// TwinCAT 3 PLC project Modbus_RTU
// ProgramVersion: 3.1.4024.12
// libraries:
//   Tc2_ModbusRTU, * (Beckhoff Automation GmbH)
//   Tc2_Standard, * (Beckhoff Automation GmbH)
//   Tc2_System, * (Beckhoff Automation GmbH)
//   Tc3_Module, * (Beckhoff Automation GmbH)
// project tree:
//   / PlcTask.TcTTO
//   POUs/ MAIN.TcPOU, P_ModbusRTU_Master.TcPOU, P_ModbusRTU_Slave.TcPOU

CONFIGURATION Modbus_RTU
    RESOURCE PLC ON TwinCAT3
        TASK PlcTask(INTERVAL := T#10ms, PRIORITY := 28);
        PROGRAM MAIN WITH PlcTask : MAIN;
    END_RESOURCE
END_CONFIGURATION

// ---- POUs/MAIN.TcPOU
PROGRAM MAIN
VAR
END_VAR

P_ModbusRTU_Master();
P_ModbusRTU_Slave();

END_PROGRAM

// ---- POUs/P_ModbusRTU_Master.TcPOU
PROGRAM P_ModbusRTU_Master
VAR
// Communication block
// ===================
	// make sure to choose the correct block depending on the type of serial port
	fbModbus		: ModbusRtuMasterV2_PcCOM;	
	//	fbModbus		: ModbusRtuMasterV2_KL6x5B;	
	//	fbModbus		: ModbusRtuMasterV2_KL6x22B;	
	
// Send and Receive data 
// =====================
	Send			: ARRAY [0..100] OF WORD;
	Rcv				: ARRAY [0..100] OF WORD;

	
// Sequence 
// ========
	bStart			: BOOL;
	Step			: INT;
END_VAR

{region "Hardware set up"}
// Linking to serial port
// ======================

// The IO's to link to the serial port are declared inside of the FB ModbusRtuMasterV2_XXXXX.
// By building/compiling the program, these IO will be generate in the PLC instance, ready to link
// This is also the reason why there are FB's for every type of serial port.

// Communication parameters serial port
// ====================================
	 
// Make sure to set up the correct communication parameters for the serial port, like:
//		* Baudrate
//		* Data bits
//		* Stop bits
//		* Xon/Xoff

// In case you are using an EL terminal, please set these CoE Online parameters:
//		* 	8000:05		"Enable transfer rate opmitization"		--> FALSE
//		*	8000:06		"Enable half duplex"					--> FALSE		(if 4 wires are used for RS485)
//																--> TRUE		(if 2 wires are used for RS485)	 

{endregion}

// Communication block
// ===================

// The communication block itself does not need to be called.
// Depending on the wanted action (read registers, read input registers, write registeres, ...), the corresponding action will be called.
// But since all these actions use the inputs/outputs from the FB itself, it is recommended to use a sequence for calling the actions


// Sequence
// ========

CASE Step OF
	0:		// Wait for start
		IF bStart THEN
			Step := 100;
		END_IF
	100:	// Read input registers 4 - 9 (so 6 modbus registers), from device address 10
		fbModbus.ReadInputRegs(Execute		:= FALSE);		// call actions with "Execute := FALSE", to be sure to have a positive edge to trigger the reading	
		fbModbus.ReadInputRegs(
			UnitID		:= 10, 
			Quantity	:= 6, 
			MBAddr		:= 4,		// Keep in mind that for some devices you have to substract 1 from the register.
			cbLength	:= SIZEOF(Rcv), 
			pMemoryAddr	:= ADR(Rcv), 
			Execute		:= TRUE, 
			Timeout		:= T#100MS,	// Always insert a time out, otherwise a time of 0ms will be used, resulting in a time out  
			BUSY		=> , 
			Error		=> , 
			ErrorId		=> , 
			cbRead		=> );
		
		IF fbModbus.BUSY THEN
			Step := 110;
		END_IF

	110:
		IF NOT fbModbus.BUSY THEN
			IF fbModbus.Error THEN
				// Code to be done in case of an error reading data, f.e.:
				Step := 100;	// if you want to try again
				Step := 0;		// if you want to retry the complete cycle
			ELSE
				// Code to be done in case of no error reading data, f.e.:
				
				// Decode received data
				// Since modbus as a standard only has words, data can be converted to store them in words.
				// for esample, reals are sometimes stored in the words by multiplying them by 10 or by 100, depeding on the wanted resolution
				
				// Reg4Value := Rcv[0] * 0.1;
				// Reg5Value := Rcv[0] * 0.01;
				// Reg6Value := Rcv[0] * 2;
				// Reg7Value := Rcv[0] * 0.1;
				// Reg8Value := Rcv[0] * 0.1;
				// Reg9Value := Rcv[0] * 0.1;
				
				Step := 200;
			END_IF
		END_IF

	200:	// Read registers 12 - 15 (so 4 modbus registers), from device address 15
		fbModbus.ReadRegs(Execute		:= FALSE);		// call actions with "Execute := FALSE", to be sure to have a positive edge to trigger the reading	
		fbModbus.ReadRegs(
			UnitID		:= 15, 
			Quantity	:= 4, 
			MBAddr		:= 12,		// Keep in mind that for some devices you have to substract 1 from the register.
			cbLength	:= SIZEOF(Rcv), 
			pMemoryAddr	:= ADR(Rcv), 
			Execute		:= TRUE, 
			Timeout		:= T#100MS,	// Always insert a time out, otherwise a time of 0ms will be used, resulting in a time out  
			BUSY		=> , 
			Error		=> , 
			ErrorId		=> , 
			cbRead		=> );
		
		IF fbModbus.BUSY THEN
			Step := 210;
		END_IF

	210:
		IF NOT fbModbus.BUSY THEN
			IF fbModbus.Error THEN
				// Code to be done in case of an error reading data, f.e.:
				Step := 200;	// if you want to try again
				Step := 0;		// if you want to retry the complete cycle
			ELSE
				// Code to be done in case of no error reading data, f.e.:
				
				// Decode received data
				// Since modbus as a standard only has words, data can be converted to store them in words.
				// for esample, reals are sometimes stored in the words by multiplying them by 10 or by 100, depeding on the wanted resolution
				
				// Reg12Value := Rcv[0] * 0.1;
				// Reg13Value := Rcv[0] * 0.01;
				// Reg14Value := Rcv[0] * 2;
				// Reg15Value := Rcv[0] * 0.1;
				
				Step := 300;
			END_IF
		END_IF

	300:	// Write registers 25 - 34 (so 10 modbus registers), to device address 27

		// fill data to send:
		Send[0]	:= 1254;		// Data for modbus register 25
		Send[1]	:= 751;			// Data for modbus register 26
		Send[2]	:= 2300;		// Data for modbus register 27
		Send[3]	:= 254;			// Data for modbus register 28
		Send[5]	:= 128;			// Data for modbus register 29
		Send[5]	:= 775;			// Data for modbus register 30
		Send[6]	:= 943;			// Data for modbus register 31
		Send[7]	:= 225;			// Data for modbus register 32
		Send[8].0	:= TRUE;	// Data for modbus register 33
		Send[8].1	:= TRUE;	// Data for modbus register 33
		Send[8].2	:= TRUE;	// Data for modbus register 33
		Send[8].5	:= TRUE;	// Data for modbus register 33
		Send[8].7	:= TRUE;	// Data for modbus register 33
		Send[9]	:= 567;			// Data for modbus register 34
 	
		fbModbus.WriteRegs(Execute		:= FALSE);		// call actions with "Execute := FALSE", to be sure to have a positive edge to trigger the reading	
		fbModbus.WriteRegs(
			UnitID		:= 27, 
			Quantity	:= 10, 
			MBAddr		:= 25,		// Keep in mind that for some devices you have to substract 1 from the register.
			cbLength	:= SIZEOF(Send), 
			pMemoryAddr	:= ADR(Send), 
			Execute		:= TRUE, 
			Timeout		:= T#100MS,	// Always insert a time out, otherwise a time of 0ms will be used, resulting in a time out  
			BUSY		=> , 
			Error		=> , 
			ErrorId		=> , 
			cbRead		=> );
		
		IF fbModbus.BUSY THEN
			Step := 310;
		END_IF

	310:
		IF NOT fbModbus.BUSY THEN
			IF fbModbus.Error THEN
				// Code to be done in case of an error reading data, f.e.:
				Step := 300;	// if you want to try again
				Step := 0;		// if you want to retry the complete cycle
			ELSE
				// Code to be done in case of no error reading data, f.e.:
				
				Step := 0;		// Return to first step
			END_IF
		END_IF
END_CASE

END_PROGRAM

// ---- POUs/P_ModbusRTU_Slave.TcPOU
PROGRAM P_ModbusRTU_Slave
VAR
// Communication block
// ===================
	// make sure to choose the correct block depending on the type of serial port
	fbModbus			: ModbusRtuSlave_PcCOM;	
	//	fbModbus		: ModbusRtuSlave_KL6x5B;	
	//	fbModbus		: ModbusRtuSlave_KL6x22B;	
	
	
// Definition of Modbus data access areas
// ======================================
	// Check the following options *)

	// hardware independent access to the input, output and memory area
	// The ranges are declared with a length of only one word
	// Nevertheless ModbusRTU will access the full length defined above

	(*
	Inputs 	AT %IW0:	WORD;
	Outputs AT %QW0:	WORD;
	Memory 	AT %MW0:	WORD;
	*)

	// The ranges are declared as arrays here (optional)
	Inputs 	AT %IW0:	ARRAY[0..255] OF WORD;
	Outputs AT %QW0:	ARRAY[0..255] OF WORD;
	Memory 	AT %MW0:	ARRAY[0..2047] OF WORD;

	// hardware independent access to normal variables
	// (no input, ouput or memory range)
	
	(*
	Inputs	:	ARRAY[0..255] OF WORD;
	Outputs :	ARRAY[0..255] OF WORD;
	Memory 	:	ARRAY[0..255] OF WORD;
	*)

END_VAR

{region "Hardware set up"}
// Linking to serial port
// ======================

// The IO's to link to the serial port are declared inside of the FB ModbusRtuMasterV2_XXXXX.
// By building/compiling the program, these IO will be generate in the PLC instance, ready to link
// This is also the reason why there are FB's for every type of serial port.

// Communication parameters serial port
// ====================================
	 
// Make sure to set up the correct communication parameters for the serial port, like:
//		* Baudrate
//		* Data bits
//		* Stop bits
//		* Xon/Xoff

// In case you are using an EL terminal, please set these CoE Online parameters:
//		* 	8000:05		"Enable transfer rate opmitization"		--> FALSE
//		*	8000:06		"Enable half duplex"					--> FALSE		(if 4 wires are used for RS485)
//																--> TRUE		(if 2 wires are used for RS485)	 

{endregion}

// Communication block
// ===================
	// Device Address is 17
	fbModbus(
		UnitID			:= 17, 
		AdrInputs		:= ADR(Inputs), 
		SizeInputBytes	:= SIZEOF(Inputs), 
		AdrOutputs		:= ADR(Outputs), 
		SizeOutputBytes	:= SIZEOF(Outputs), 
		AdrMemory		:= ADR(Memory), 
		SizeMemoryBytes	:= SIZEOF(Memory), 
		ErrorId			=> );

END_PROGRAM
